# EPICS substitutions: vmemon/snmpApp/Db/MitsubishiUPS.substitutions
# Mitsubishi UPS file
#Test Utility Commands
#snmpwalk -Os -c public -v 1 10.0.145.033 1.3.6.1.4.1.13891.101.2
#snmpget -v 1 -c public 10.0.145.033 1.3.6.1.4.1.13891.101.2
#sudo -E wireshark
#
file "MitsubishiUPSsnmp.template"
{

     pattern { Pri,               Sec,        Dev,      Assembly,    Scan,          C,         IP,               Dev_N,    Sec_N,                    Flnk}

	    { "CF:CmptrRm",      ":CR",       "{UPS:3}",   "",     "10 second",     "public",    "10.0.145.33",          "",           "",         ""         }

}
